// TIA Portal V20 export
DATA_BLOCK "InstProfinetDeviceDiagStatus"   // DB215
// stored: InstanceOfName LER_DiagnosticsStatus, InstanceOfType FB
"LER_DiagnosticsStatus"
   // VAR_INPUT
   //    devStateHmi_X1 : Array[0..256] of "LAF_typeDevDiagBasic";
   //    devStateHmi_X2 : Array[0..256] of "LAF_typeDevDiagBasic";
   //    UnitSelect : Int := 3;
   //    Reset : Bool := FALSE;
   // END_VAR
   // VAR_IN_OUT
   //    DevState : "LER_DiagnosticsInterface";
   // END_VAR
   // VAR
   //    staticCntState : Int := 189;
   //    staticCntStartState : Int := 1;
   //    staticCntEndState : Int := 200;
   //    staticCntDev : Int := 5;
   //    staticCntHighLimit_X2 : Array[1..15] of Int;
   //    staticCntLowLimit_X2 : Array[1..15] of Int;
   //    staticCntHighLimit_X1 : Array[1..15] of Int;
   //    staticCntLowLimit_X1 : Array[1..15] of Int;
   //    staticCntModuleState : Int := 69;
   //    staticDevStateError : Array[0..15] of Bool;
   //    statiDevStateMove_X1 : Array[0..15] of Int;
   //    statiDevStateMove_X2 : Array[0..15] of Int;
   // END_VAR
BEGIN
   devStateHmi_X1[0..256].devNumber := 0;
   devStateHmi_X1[0..256].devName := '';
   devStateHmi_X1[0..256].devStateDezCoded := 0;
   devStateHmi_X1[0..256].devStateBitCoded := 16#0000;
   devStateHmi_X1[0..256].first8CharOfMlfb := '';
   devStateHmi_X2[0..256].devNumber := 0;
   devStateHmi_X2[0..256].devName := '';
   devStateHmi_X2[0..256].devStateDezCoded := 0;
   devStateHmi_X2[0..256].devStateBitCoded := 16#0000;
   devStateHmi_X2[0..256].first8CharOfMlfb := '';
   staticCntHighLimit_X2[1] := 2;
   staticCntHighLimit_X2[2] := 33;
   staticCntHighLimit_X2[3] := 42;
   staticCntHighLimit_X2[4] := 68;
   staticCntHighLimit_X2[5] := 91;
   staticCntHighLimit_X2[6] := 115;
   staticCntHighLimit_X2[7] := 133;
   staticCntHighLimit_X2[8] := 143;
   staticCntHighLimit_X2[9] := 170;
   staticCntHighLimit_X2[10..15] := 0;
   staticCntLowLimit_X2[1] := 2;
   staticCntLowLimit_X2[2] := 30;
   staticCntLowLimit_X2[3] := 42;
   staticCntLowLimit_X2[4] := 61;
   staticCntLowLimit_X2[5] := 81;
   staticCntLowLimit_X2[6] := 101;
   staticCntLowLimit_X2[7] := 121;
   staticCntLowLimit_X2[8] := 141;
   staticCntLowLimit_X2[9] := 161;
   staticCntLowLimit_X2[10..15] := 0;
   staticCntHighLimit_X1[1] := 1;
   staticCntHighLimit_X1[2] := 29;
   staticCntHighLimit_X1[3] := 41;
   staticCntHighLimit_X1[4..15] := 0;
   staticCntLowLimit_X1[1] := 1;
   staticCntLowLimit_X1[2] := 21;
   staticCntLowLimit_X1[3] := 41;
   staticCntLowLimit_X1[4..15] := 0;
   staticDevStateError[0..15] := FALSE;
   statiDevStateMove_X1[0] := 0;
   statiDevStateMove_X1[1] := 1;
   statiDevStateMove_X1[2] := 9;
   statiDevStateMove_X1[3] := 1;
   statiDevStateMove_X1[4..15] := 0;
   statiDevStateMove_X2[0] := 0;
   statiDevStateMove_X2[1] := 2;
   statiDevStateMove_X2[2] := 13;
   statiDevStateMove_X2[3] := 2;
   statiDevStateMove_X2[4] := 8;
   statiDevStateMove_X2[5] := 11;
   statiDevStateMove_X2[6] := 15;
   statiDevStateMove_X2[7] := 13;
   statiDevStateMove_X2[8] := 3;
   statiDevStateMove_X2[9] := 10;
   statiDevStateMove_X2[10..15] := 0;
END_DATA_BLOCK
